(* IEC 61131-3 sources: SRCI/RobotLibrary/RobotLibrary/POUs/Write/MC_WriteLoadData, 1 file *)

(* ---- MC_WriteLoadDataFB.st ---- *)
/// Change configuration of selected payload number
FUNCTION_BLOCK MC_WriteLoadDataFB EXTENDS RobotLibraryBaseExecuteFB
// -------------------------------------------------------------------------
//  SRCI Robot Library
// -------------------------------------------------------------------------
//
//  Object:      WriteLoadDataFB
//  Author:      Thorsten Brach
//  Date:        2024-06-01
//
//  Description:
//
//
//  Copyright:
//    (C) 2024 Thorsten Brach. All rights reserved
//             Licensed under the LGPL-3.0 license.
//
//  Disclaimer:
//    This project is provided without any guarantee and can be used for
//    private and commercial purposes. Any use is at the user’s
//    own risk and responsibility.
//
// -------------------------------------------------------------------------
VAR_INPUT
  /// Defines the target sequence in which the command will be executed
  SequenceFlag       : SequenceFlag;
  /// Processing Mode
  ProcessingMode     : ProcessingMode;
  /// command parameter
  ParCmd             : WriteLoadDataParCmd;
END_VAR
VAR_OUTPUT
  /// Command is transferred and confirmed by the RC
  CommandBuffered    : BOOL;
  /// The command was aborted by another command
  CommandAborted     : BOOL;
  /// TRUE, while command is interrupted during execution and can be continued.
  CommandInterrupted : BOOL;
  /// command outputs
  OutCmd             : WriteLoadDataOutCmd;
END_VAR

VAR
  /// internal copy of command parameter
 _parCmd             : WriteLoadDataParCmd;
  /// command data to send
 _command            : WriteLoadDataSendData;
  /// response data received
 _response           : WriteLoadDataRecvData;
END_VAR

  SUPER^(AxesGroup := AxesGroup);

END_FUNCTION_BLOCK

METHOD CheckParameterChanged : BOOL
VAR_IN_OUT
  /// Robot assignment of function
  AxesGroup    : AxesGroup;
END_VAR

  // Check ParCmd Size is > 0, becaue MemCmp does not work correctly with size = 0
  IF (SIZEOF(ParCmd) = 0)
  THEN
    RETURN;
  END_IF

  // compare memory
  CheckParameterChanged := ( MemCmp(ADR(ParCmd), ADR(_parCmd), SIZEOF(ParCmd)) <> RobotLibraryConstants.OK );

  IF ( CheckParameterChanged )
  THEN
    // update internal copy of parameters
   _parCmd := ParCmd;
    // inc parameter sequence
   _command.ParSeq := _command.ParSeq + 1;
    // update command data
    CommandData := CreateCommandPayload(); // ( Access via reference to rCommandFB in ACR )
    // notify active command register
    AxesGroup.Acyclic.ActiveCommandRegister.NotifyParameterChanged := _uniqueID;
  END_IF

END_METHOD

METHOD INTERNAL CreateCommandPayload : SendData
// Table 6-132: Sent CMD payload (PLC to RC) of "WriteLoadData"
// --------------------------
// Header
// --------------------------
// Byte 00 : UINT  - Type HB
// Byte 01 :       - Type LB
// Byte 02 : USINT - Reserve | ExecutionMode
// Byte 03 : USINT - ParSeq  | Priority
// --------------------------
// Datablock
// --------------------------
// Byte 04 : DATE LoadData.Date
// Byte 05 :
// Byte 06 : TIME_OF_DAY LoadData.Time
// Byte 07 :
// Byte 08 :
// Byte 09 : REAL LoadData.X
// Byte 10 :
// Byte 11 :
// Byte 12 :
// Byte 13 : REAL LoadData.Y
// Byte 14 :
// Byte 15 :
// Byte 16 :
// Byte 17 : REAL LoadData.Z
// Byte 18 :
// Byte 19 :
// Byte 20 :
// Byte 21 : REAL LoadData.RX
// Byte 22 :
// Byte 23 :
// Byte 24 :
// Byte 25 : REAL LoadData.RY
// Byte 26 :
// Byte 27 :
// Byte 28 :
// Byte 29 : REAL LoadData.RZ
// Byte 30 :
// Byte 31 :
// Byte 32 :
// Byte 33 : REAL LoadData.Mass
// Byte 34 :
// Byte 35 :
// Byte 36 :
// Byte 37 : REAL LoadData.IX
// Byte 38 :
// Byte 39 :
// Byte 40 :
// Byte 41 : REAL LoadData.IY
// Byte 42 :
// Byte 43 :
// Byte 44 :
// Byte 45 : REAL LoadData.IZ
// Byte 46 :
// Byte 47 :
// Byte 48 :
// Byte 49 : USINT LoadNo
// --------------------------

  // set command parameter
  _command.CmdTyp   :=  CmdType.WriteLoadData;
  _command.ExecMode :=  ExecMode;
  _command.ParSeq   := _command.ParSeq;
  _command.Priority :=  Priority;
  _command.LoadData := _parCmd.LoadData;
  _command.LoadNo   := _parCmd.LoadNo;

  // copy command data to header
  _cmdHeader := _command;
  // call base implementation to copy header to payload buffer
  CreateCommandPayload := SUPER^.CreateCommandPayload();

  // add command.LoadData.Timestamp.IEC_DATE
  CreateCommandPayload.AddUint(_command.LoadData.Timestamp.IEC_DATE);
  // add command.LoadData.Timestamp.IEC_TIME
  CreateCommandPayload.AddTime(_command.LoadData.Timestamp.IEC_TIME);
  // add command.LoadData.X
  CreateCommandPayload.AddReal(_command.LoadData.X);
  // add command.LoadData.Y
  CreateCommandPayload.AddReal(_command.LoadData.Y);
  // add command.LoadData.Z
  CreateCommandPayload.AddReal(_command.LoadData.Z);
  // add command.LoadData.Rx
  CreateCommandPayload.AddReal(_command.LoadData.Rx);
  // add command.LoadData.Ry
  CreateCommandPayload.AddReal(_command.LoadData.Ry);
  // add command.LoadData.Rz
  CreateCommandPayload.AddReal(_command.LoadData.Rz);
  // add command.LoadData.Mass
  CreateCommandPayload.AddReal(_command.LoadData.Mass);
  // add command.LoadData.Ix
  CreateCommandPayload.AddReal(_command.LoadData.Ix);
  // add command.LoadData.Iy
  CreateCommandPayload.AddReal(_command.LoadData.Iy);
  // add command.LoadData.Iz
  CreateCommandPayload.AddReal(_command.LoadData.Iz);
  // add command.LoadNo
  CreateCommandPayload.AddUsint(_command.LoadNo);

END_METHOD

METHOD FB_init : BOOL
VAR_INPUT
  /// if TRUE, the retain variables are initialized (warm start / cold start)
	bInitRetains : BOOL;
  /// if TRUE, the instance afterwards gets moved into the copy code (online change)
	bInCopyCode  : BOOL;
END_VAR

  MyType := 'MC_WriteLoadDataFB';

  ExecMode := ExecutionMode.PARALLEL;

END_METHOD

METHOD PROTECTED OnCall
VAR_IN_OUT
  /// Robot assignment of function
  AxesGroup : AxesGroup;
END_VAR

  // call base implementation
  SUPER^.OnCall(AxesGroup := AxesGroup);

  CASE _stepCmd OF

    00:  IF ( _execute_R.Q )
         THEN
           // set busy flag
           Busy := TRUE;
           // Reset command outputs
           MemSet(ADR(OutCmd),0,SIZEOF(OutCmd));
           // apply command parameter
          _parCmd := ParCmd;
           // init parameter sequence
          _command.ParSeq := 1;
           // set timeout
           SetTimeout(PT := _timeoutCmd, rTimer := _timerCmd);
           // inc step counter
          _stepCmd := _stepCmd + 1;
  	     END_IF

    01:  // create command data
         CommandData := CreateCommandPayload();
         // Add command to active command register
        _uniqueID := AxesGroup.Acyclic.ActiveCommandRegister.AddCmd( pCommandFB := ADR(THIS^ ));
         // set timeout
         SetTimeout(PT := _timeoutCmd, rTimer := _timerCmd);
         // inc step counter
        _stepCmd := _stepCmd + 1;

    02:  // Wait for responce received
         IF ( _responseReceived )
         THEN
           // reset response received flag
          _responseReceived := FALSE;

           CASE  _response.State
           OF
             CmdMessageState.BUFFERED    : CommandBuffered    := TRUE;
             CmdMessageState.ABORTED     : CommandAborted     := TRUE;
             CmdMessageState.INTERRUPTED : CommandInterrupted := TRUE;
             CmdMessageState.DONE        : Done               := TRUE;
             CmdMessageState.ERROR       : Error              := TRUE;
  				 END_CASE

           // Done, Aborted or Error ?
           IF (_response.State >= CmdMessageState.DONE )
           THEN
             // Reset Busy flag
             Busy := FALSE;
             // set timeout
             SetTimeout(PT := _timeoutCmd, rTimer := _timerCmd);
             // inc step counter
            _stepCmd := _stepCmd + 1;
  				 END_IF
         END_IF

    03: IF ( NOT Execute)
        THEN
          Reset();
  			END_IF
  ELSE
    // invalid step
    ErrorID := RobotLibraryEvents.ERR_INVALID_STEP;
  END_CASE

  // Cancel
  IF (Busy) AND (NOT Execute)
  THEN
    // try to remove cmd
    AxesGroup.Acyclic.ActiveCommandRegister.RemoveCmd(_uniqueID);
  END_IF

  // Reset FB
  IF ( NOT Execute )
  THEN
    Reset();
  END_IF

END_METHOD

METHOD INTERNAL ParseResponsePayload : DINT
// Table 6-133: Received CMD payload (RC to PLC) of "WriteLoadData"
// --------------------------
// Header
// --------------------------
// Byte 00 : USINT   - ParSeq | State
// Byte 01 : SINT    - AlarmMessageSeverity
// Byte 02 : UINT    - AlarmMessageCode HB
// Byte 03 :         - AlarmMessageCode LB
// --------------------------
// Datablock
// --------------------------
// Byte 04 : USINT      - InvocationCounter
// Byte 05 : SINT       - Reserved
// Byte 06 : INT        - OriginID HW HB
// Byte 07 :            - OriginID HW LB
VAR_INPUT
  /// Response data
  ResponseData : RecvData;
END_VAR

  // call base implementation to parse the header from payload buffer
  ResponseData.PayloadPtr := SUPER^.ParseResponsePayload(ResponseData);

  // copy parsed header to response
  _response.ParSeq               := _rspHeader.ParSeq;
  _response.State                := _rspHeader.State;
  _response.AlarmMessageSeverity := _rspHeader.AlarmMessageSeverity;
  _response.AlarmMessageCode     := _rspHeader.AlarmMessageCode;

END_METHOD

METHOD PROTECTED Reset : DINT
VAR_INPUT
END_VAR

  Reset := SUPER^.Reset();

  Done               := FALSE;
  Busy               := FALSE;
  CommandBuffered    := FALSE;
  CommandAborted     := FALSE;
  CommandInterrupted := FALSE;

END_METHOD
